{attribute 'linkalways'} 
{attribute 'no_explicit_call' := 'This FB is a CLASS and must be accessed using methods or properties'}
{attribute 'enable_dynamic_creation'}
FUNCTION_BLOCK Node_F_VN_WatershedSegmentationExp EXTENDS VisionNode
VAR
	ipSrcImage : _ITcVnImage;
    ipDestImage : _ITcVnImage;
    ipMarkers : _ITcVnImage;
    hrPrev : _HRESULT(S_OK);
	hresult : _HRESULT(S_OK);
END_VAR

METHOD PUBLIC  Clone : I_Node
VAR
	pNode : POINTER TO Node_F_VN_WatershedSegmentationExp;
END_VAR
pNode := __NEW(Node_F_VN_WatershedSegmentationExp);
Clone := pNode^;
END_METHOD

METHOD FB_init : BOOL
VAR_INPUT
	bInitRetains : BOOL; // if TRUE, the retain variables are initialized (warm start / cold start)
	bInCopyCode : BOOL;  // if TRUE, the instance afterwards gets moved into the copy code (online change)
END_VAR
AddInput('ipSrcImage', ipSrcImage);
AddInput('ipMarkers', ipMarkers);
AddInput('hrPrev', hrPrev);
AddOutput('ipDestImage', ipDestImage);
AddOutput('hresult',hresult);
END_METHOD

METHOD PROTECTED OnExecute
hresult.Value := F_VN_WatershedSegmentationExp(
	ipSrcImage := ipSrcImage.Value,
	ipDestImage := ipDestImage.Value,
    ipMarkers := ipMarkers.Value,
	hrPrev := hrPrev.Value);
END_METHOD

METHOD PUBLIC PreExecutionCheck
VAR_INPUT
	Check : I_PreExecutionChecks;
END_VAR
Check.IsTrue(ipSrcImage.IsValid, 'ipSrcImage must contain an image');
Check.IsTrue(ipSrcImage.HasChannelCount(3), 'ipSrcImage must have 3 channels');
Check.IsTrue(ipSrcImage.IsPixelDepth(8), 'ipSrcImage must have 8 bit pixel depth');
Check.IsTrue(ipMarkers.IsValid, 'ipMarkers must contain an image');
Check.IsTrue(ipMarkers.HasChannelCount(1), 'ipMarkers must have 1 channel');
Check.IsTrue(ipMarkers.IsPixelDepth(32), 'ipMarkers must have DINT 32 bit pixel depth');
END_METHOD

END_FUNCTION_BLOCK

(* stored: Version 1.1.0.1, ProductVersion 3.1.4024.15
   POU Node_F_VN_WatershedSegmentationExp: Id {4dda013b-dfc2-069e-36f5-965e7af3f489}, SpecialFunc None
   Folder Constructor: Id {127a547a-a274-0135-09ac-c3f37a04d1bd}
   Method Clone: Id {86969201-5477-0eeb-32e0-2c57fe45d285}
   Method FB_init: Id {3d97477b-7799-060a-236d-fdf4c87cb003}
   Method OnExecute: Id {ef2bd86f-ae01-001f-3624-4de04e26ca81}
   Method PreExecutionCheck: Id {6808313b-67e5-093b-1502-3a38930096e3} *)
